FUNCTION_BLOCK FB_WriteVariableByName

VAR_INPUT
	sName  : STRING;
	sValue : STRING;
	bExec  : BOOL;
END_VAR

VAR_OUTPUT
	Busy   : BOOL := FALSE;
	Error  : BOOL := FALSE;
	Done   :  BOOL := FALSE;
END_VAR

VAR
	nState 	: INT := 0;
	rtrig  	: R_TRIG;
	
	fbSymInfo		: PLC_ReadSymInfoByName := ( PORT := 851, TMOUT := DEFAULT_ADS_TIMEOUT );
  stSymbolInfo	: Tc2_Utilities.SYMINFOSTRUCT;
  fbWriteReq    : ADSWRITE := ( NETID := '', PORT := 851, TMOUT := DEFAULT_ADS_TIMEOUT );
	
	// Native variables for various datatypes that can be set in XML.
	// Depending on the type one variable is selected to receive the string conversion result.
  // The address will be used as data input of ADSWRITE-FB.
  
	var_data : ST_VARIANT; 
	
END_VAR

 
rtrig(CLK:= bExec , Q=> );

 CASE nState OF

	0:	// Wait for request
		IF (NOT bExec) THEN
			error := FALSE; done := FALSE;
		END_IF

		IF (rtrig.Q) THEN
			Busy:= TRUE;
			nState:= nState + 1;
		END_IF

	1:
		// reset FB
		IF (fbSymInfo.START AND NOT fbSymInfo.BUSY) THEN
			fbSymInfo( START:= FALSE);
		END_IF
		// get symbol information
		fbSymInfo
    ( 
		 	symname := sName,
	   	syminfo => stSymbolInfo,
	   	start:= TRUE
		);
		// 
		IF (NOT fbSymInfo.BUSY) THEN
	 	  IF (fbSymInfo.ERR) THEN
				nState := 99;
		  ELSE
				IF (F_ParseToVariant (adsTypeID:= stSymbolInfo.adsDataType,
							                sValue:= sValue, var_data:= var_data))
				THEN
					nState := nState + 1;
				ELSE
					nState := 99;
				END_IF
		  END_IF
		END_IF
		
	2:	// write the value
		
		// reset FB
		IF (fbWriteReq.WRITE AND NOT fbWriteReq.BUSY) THEN
			fbWriteReq(WRITE := FALSE);
		END_IF
		// write variable
		fbWriteReq
		(
			IDXGRP:= stSymbolInfo.idxGroup, 
			IDXOFFS:= stSymbolInfo.idxOffset,
			SRCADDR := ADR(var_data),
			LEN := stSymbolInfo.byteSize,
			WRITE := TRUE 
		);
		IF (NOT fbWriteReq.BUSY) THEN
	 		IF (fbWriteReq.ERR) THEN
			  nState := 99;
			ELSE
			  nState := 100;
			END_IF
		END_IF
	
	99:	// Error
		busy := FALSE;
		error := TRUE;
		nState := 0;
				
	100: // Success
		busy := FALSE;
		done := TRUE;
		nState := 0;
 
 END_CASE

END_FUNCTION_BLOCK

(* stored: Version 1.1.0.1, ProductVersion 3.1.4024.12
   POU FB_WriteVariableByName: Id {f0cbcd71-a206-42a6-9949-9cd5a3db7fae}, SpecialFunc None *)
